% RSLogix 500 project Villa_Park_Riverside_Dump_SLC_500_April_16_2021.RSS, saved by version 11.00.00.00 %
PROJECT "AIRDROME"    % processor: type code 8 %

PROGRAM FILES
  LAD 2   52 rungs

DATA FILES
  O0 OUTPUT  2 elements
  I1 INPUT  3 elements
  S2 STATUS  16 elements
  B3 BINARY  3 elements
  T4 TIMER  15 elements
  C5 COUNTER  1 elements
  R6 CONTROL  1 elements
  N7 INTEGER  1 elements

LADDER 2
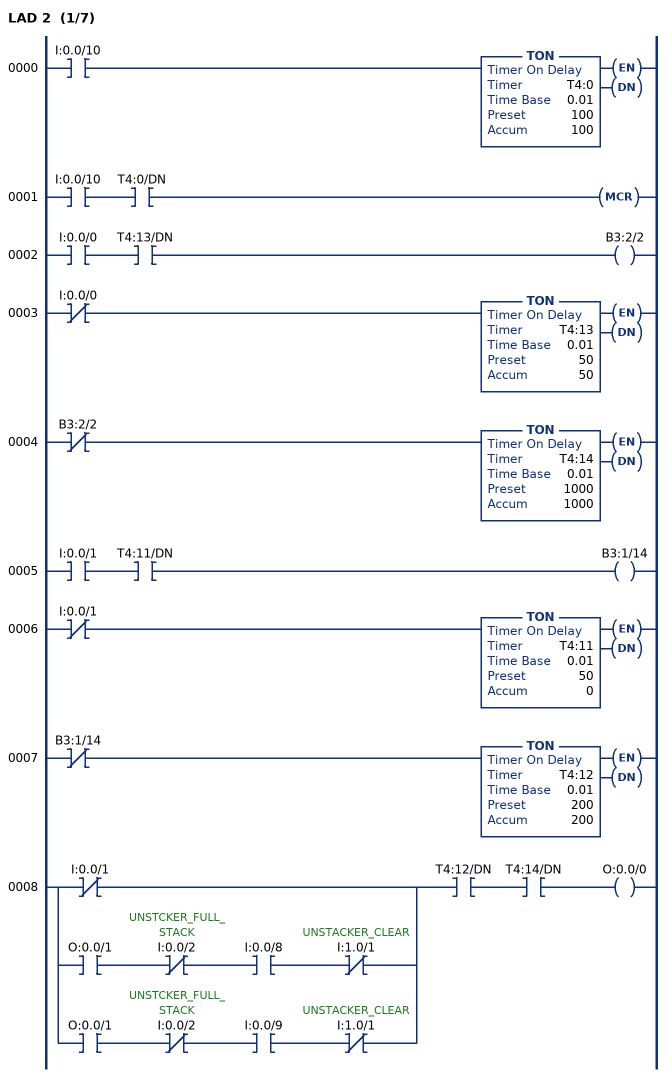
% Rung: 0 %
SOR XIC I:0.0/10 TON T4:0 0.01 100 100 EOR
% Rung: 1 %
SOR XIC I:0.0/10 XIC T4:0/DN MCR EOR
% Rung: 2 %
SOR XIC I:0.0/0 XIC T4:13/DN OTE B3:2/2 EOR
% Rung: 3 %
SOR XIO I:0.0/0 TON T4:13 0.01 50 50 EOR
% Rung: 4 %
SOR XIO B3:2/2 TON T4:14 0.01 1000 1000 EOR
% Rung: 5 %
SOR XIC I:0.0/1 XIC T4:11/DN OTE B3:1/14 EOR
% Rung: 6 %
SOR XIO I:0.0/1 TON T4:11 0.01 50 0 EOR
% Rung: 7 %
SOR XIO B3:1/14 TON T4:12 0.01 200 200 EOR
% Rung: 8 %
SOR BST XIO I:0.0/1 NXB XIC O:0.0/1 XIO I:0.0/2 XIC I:0.0/8 XIO I:1.0/1 NXB XIC O:0.0/1 XIO I:0.0/2 XIC I:0.0/9 XIO I:1.0/1 BND XIC T4:12/DN XIC T4:14/DN OTE O:0.0/0 EOR
%   I:0.0/2  UNSTCKER_FULL_STACK %
%   I:1.0/1  UNSTACKER_CLEAR %

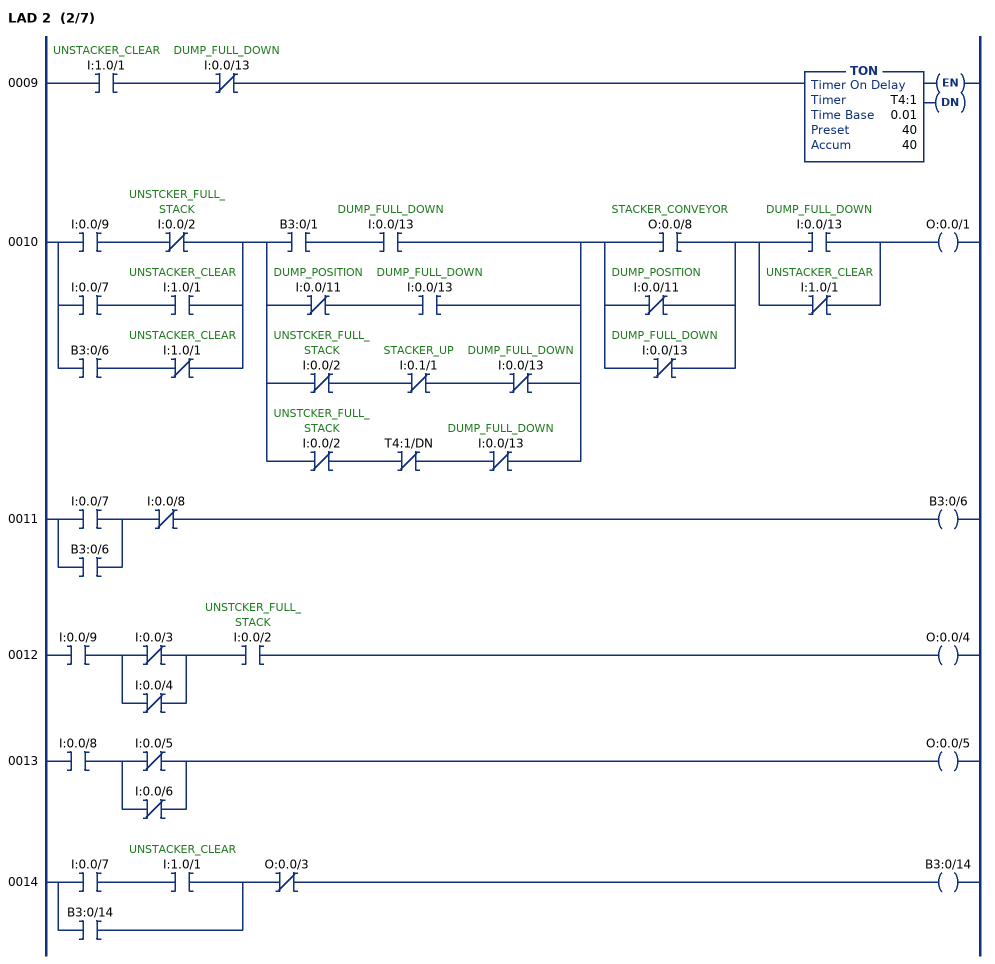
% Rung: 9 %
SOR XIC I:1.0/1 XIO I:0.0/13 TON T4:1 0.01 40 40 EOR
%   I:1.0/1  UNSTACKER_CLEAR %
%   I:0.0/13  DUMP_FULL_DOWN %
% Rung: 10 %
SOR BST XIC I:0.0/9 XIO I:0.0/2 NXB XIC I:0.0/7 XIC I:1.0/1 NXB XIC B3:0/6 XIO I:1.0/1 BND BST XIC B3:0/1 XIC I:0.0/13 NXB XIO I:0.0/11 XIC I:0.0/13 NXB XIO I:0.0/2 XIO I:0.1/1 XIO I:0.0/13 NXB XIO I:0.0/2 XIO T4:1/DN XIO I:0.0/13 BND BST XIC O:0.0/8 NXB XIO I:0.0/11 NXB XIO I:0.0/13 BND BST XIC I:0.0/13 NXB XIO I:1.0/1 BND OTE O:0.0/1 EOR
%   I:0.0/2  UNSTCKER_FULL_STACK %
%   I:1.0/1  UNSTACKER_CLEAR %
%   I:0.0/13  DUMP_FULL_DOWN %
%   I:0.0/11  DUMP_POSITION %
%   I:0.1/1  STACKER_UP %
%   O:0.0/8  STACKER_CONVEYOR %
% Rung: 11 %
SOR BST XIC I:0.0/7 NXB XIC B3:0/6 BND XIO I:0.0/8 OTE B3:0/6 EOR
% Rung: 12 %
SOR XIC I:0.0/9 BST XIO I:0.0/3 NXB XIO I:0.0/4 BND XIC I:0.0/2 OTE O:0.0/4 EOR
%   I:0.0/2  UNSTCKER_FULL_STACK %
% Rung: 13 %
SOR XIC I:0.0/8 BST XIO I:0.0/5 NXB XIO I:0.0/6 BND OTE O:0.0/5 EOR
% Rung: 14 %
SOR BST XIC I:0.0/7 XIC I:1.0/1 NXB XIC B3:0/14 BND XIO O:0.0/3 OTE B3:0/14 EOR
%   I:1.0/1  UNSTACKER_CLEAR %

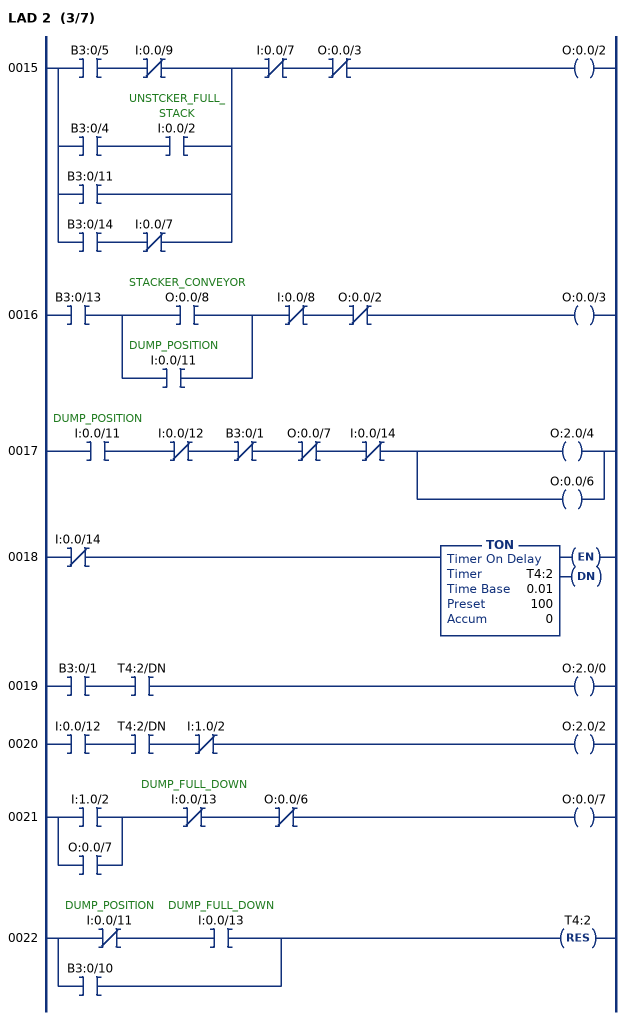
% Rung: 15 %
SOR BST XIC B3:0/5 XIO I:0.0/9 NXB XIC B3:0/4 XIC I:0.0/2 NXB XIC B3:0/11 NXB XIC B3:0/14 XIO I:0.0/7 BND XIO I:0.0/7 XIO O:0.0/3 OTE O:0.0/2 EOR
%   I:0.0/2  UNSTCKER_FULL_STACK %
% Rung: 16 %
SOR XIC B3:0/13 BST XIC O:0.0/8 NXB XIC I:0.0/11 BND XIO I:0.0/8 XIO O:0.0/2 OTE O:0.0/3 EOR
%   O:0.0/8  STACKER_CONVEYOR %
%   I:0.0/11  DUMP_POSITION %
% Rung: 17 %
SOR XIC I:0.0/11 XIO I:0.0/12 XIO B3:0/1 XIO O:0.0/7 XIO I:0.0/14 BST OTE O:2.0/4 NXB OTE O:0.0/6 BND EOR
%   I:0.0/11  DUMP_POSITION %
% Rung: 18 %
SOR XIO I:0.0/14 TON T4:2 0.01 100 0 EOR
% Rung: 19 %
SOR XIC B3:0/1 XIC T4:2/DN OTE O:2.0/0 EOR
% Rung: 20 %
SOR XIC I:0.0/12 XIC T4:2/DN XIO I:1.0/2 OTE O:2.0/2 EOR
% Rung: 21 %
SOR BST XIC I:1.0/2 NXB XIC O:0.0/7 BND XIO I:0.0/13 XIO O:0.0/6 OTE O:0.0/7 EOR
%   I:0.0/13  DUMP_FULL_DOWN %
% Rung: 22 %
SOR BST XIO I:0.0/11 XIC I:0.0/13 NXB XIC B3:0/10 BND RES T4:2 EOR
%   I:0.0/11  DUMP_POSITION %
%   I:0.0/13  DUMP_FULL_DOWN %

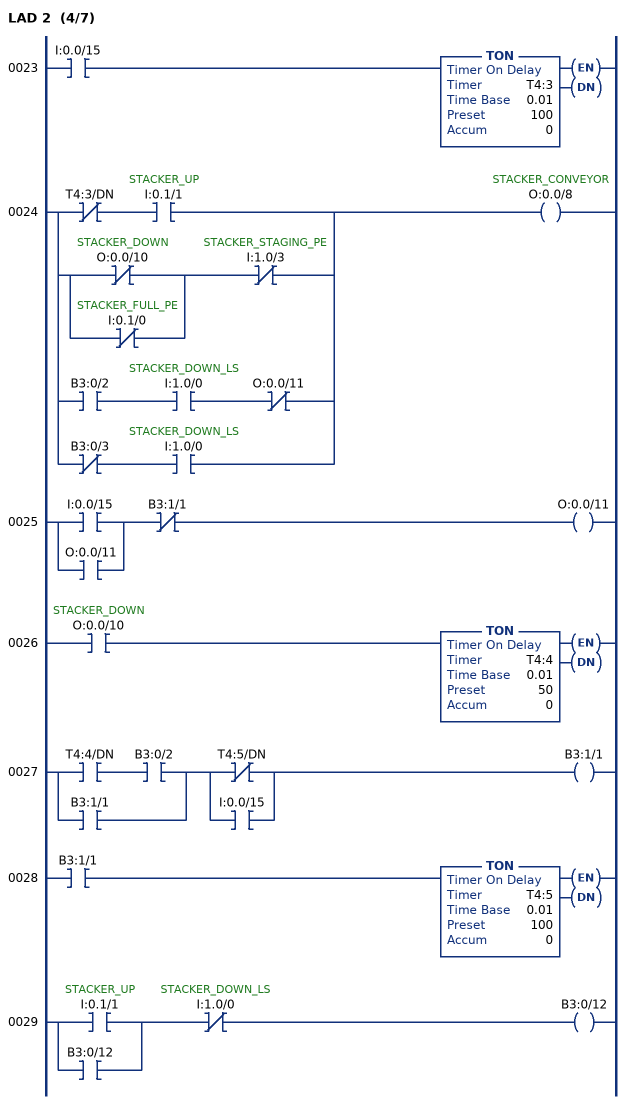
% Rung: 23 %
SOR XIC I:0.0/15 TON T4:3 0.01 100 0 EOR
% Rung: 24 %
SOR BST BST XIO T4:3/DN XIC I:0.1/1 NXB BST XIO O:0.0/10 NXB XIO I:0.1/0 BND XIO I:1.0/3 BND NXB XIC B3:0/2 XIC I:1.0/0 XIO O:0.0/11 NXB XIO B3:0/3 XIC I:1.0/0 BND OTE O:0.0/8 EOR
%   I:0.1/1  STACKER_UP %
%   O:0.0/10  STACKER_DOWN %
%   I:0.1/0  STACKER_FULL_PE %
%   I:1.0/3  STACKER_STAGING_PE %
%   I:1.0/0  STACKER_DOWN_LS %
%   O:0.0/8  STACKER_CONVEYOR %
% Rung: 25 %
SOR BST XIC I:0.0/15 NXB XIC O:0.0/11 BND XIO B3:1/1 OTE O:0.0/11 EOR
% Rung: 26 %
SOR XIC O:0.0/10 TON T4:4 0.01 50 0 EOR
%   O:0.0/10  STACKER_DOWN %
% Rung: 27 %
SOR BST XIC T4:4/DN XIC B3:0/2 NXB XIC B3:1/1 BND BST XIO T4:5/DN NXB XIC I:0.0/15 BND OTE B3:1/1 EOR
% Rung: 28 %
SOR XIC B3:1/1 TON T4:5 0.01 100 0 EOR
% Rung: 29 %
SOR BST XIC I:0.1/1 NXB XIC B3:0/12 BND XIO I:1.0/0 OTE B3:0/12 EOR
%   I:0.1/1  STACKER_UP %
%   I:1.0/0  STACKER_DOWN_LS %

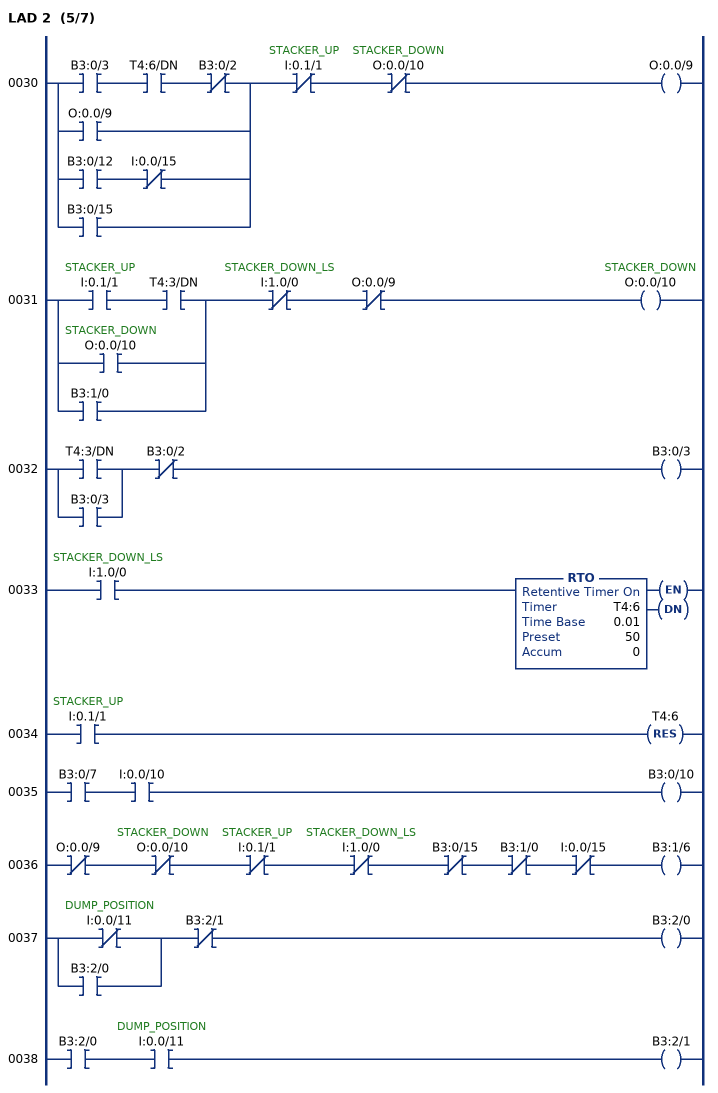
% Rung: 30 %
SOR BST XIC B3:0/3 XIC T4:6/DN XIO B3:0/2 NXB XIC O:0.0/9 NXB XIC B3:0/12 XIO I:0.0/15 NXB XIC B3:0/15 BND XIO I:0.1/1 XIO O:0.0/10 OTE O:0.0/9 EOR
%   I:0.1/1  STACKER_UP %
%   O:0.0/10  STACKER_DOWN %
% Rung: 31 %
SOR BST XIC I:0.1/1 XIC T4:3/DN NXB XIC O:0.0/10 NXB XIC B3:1/0 BND XIO I:1.0/0 XIO O:0.0/9 OTE O:0.0/10 EOR
%   I:0.1/1  STACKER_UP %
%   O:0.0/10  STACKER_DOWN %
%   I:1.0/0  STACKER_DOWN_LS %
% Rung: 32 %
SOR BST XIC T4:3/DN NXB XIC B3:0/3 BND XIO B3:0/2 OTE B3:0/3 EOR
% Rung: 33 %
SOR XIC I:1.0/0 RTO T4:6 0.01 50 0 EOR
%   I:1.0/0  STACKER_DOWN_LS %
% Rung: 34 %
SOR XIC I:0.1/1 RES T4:6 EOR
%   I:0.1/1  STACKER_UP %
% Rung: 35 %
SOR XIC B3:0/7 XIC I:0.0/10 OTE B3:0/10 EOR
% Rung: 36 %
SOR XIO O:0.0/9 XIO O:0.0/10 XIO I:0.1/1 XIO I:1.0/0 XIO B3:0/15 XIO B3:1/0 XIO I:0.0/15 OTE B3:1/6 EOR
%   O:0.0/10  STACKER_DOWN %
%   I:0.1/1  STACKER_UP %
%   I:1.0/0  STACKER_DOWN_LS %
% Rung: 37 %
SOR BST XIO I:0.0/11 NXB XIC B3:2/0 BND XIO B3:2/1 OTE B3:2/0 EOR
%   I:0.0/11  DUMP_POSITION %
% Rung: 38 %
SOR XIC B3:2/0 XIC I:0.0/11 OTE B3:2/1 EOR
%   I:0.0/11  DUMP_POSITION %

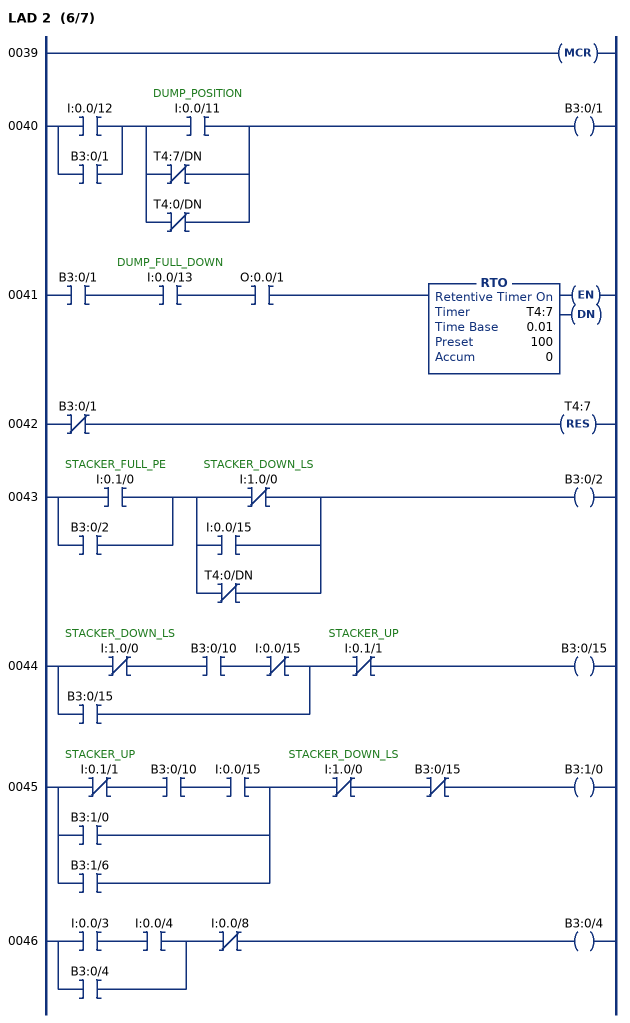
% Rung: 39 %
SOR MCR EOR
% Rung: 40 %
SOR BST XIC I:0.0/12 NXB XIC B3:0/1 BND BST XIC I:0.0/11 NXB XIO T4:7/DN NXB XIO T4:0/DN BND OTE B3:0/1 EOR
%   I:0.0/11  DUMP_POSITION %
% Rung: 41 %
SOR XIC B3:0/1 XIC I:0.0/13 XIC O:0.0/1 RTO T4:7 0.01 100 0 EOR
%   I:0.0/13  DUMP_FULL_DOWN %
% Rung: 42 %
SOR XIO B3:0/1 RES T4:7 EOR
% Rung: 43 %
SOR BST XIC I:0.1/0 NXB XIC B3:0/2 BND BST XIO I:1.0/0 NXB XIC I:0.0/15 NXB XIO T4:0/DN BND OTE B3:0/2 EOR
%   I:0.1/0  STACKER_FULL_PE %
%   I:1.0/0  STACKER_DOWN_LS %
% Rung: 44 %
SOR BST XIO I:1.0/0 XIC B3:0/10 XIO I:0.0/15 NXB XIC B3:0/15 BND XIO I:0.1/1 OTE B3:0/15 EOR
%   I:1.0/0  STACKER_DOWN_LS %
%   I:0.1/1  STACKER_UP %
% Rung: 45 %
SOR BST XIO I:0.1/1 XIC B3:0/10 XIC I:0.0/15 NXB XIC B3:1/0 NXB XIC B3:1/6 BND XIO I:1.0/0 XIO B3:0/15 OTE B3:1/0 EOR
%   I:0.1/1  STACKER_UP %
%   I:1.0/0  STACKER_DOWN_LS %
% Rung: 46 %
SOR BST XIC I:0.0/3 XIC I:0.0/4 NXB XIC B3:0/4 BND XIO I:0.0/8 OTE B3:0/4 EOR

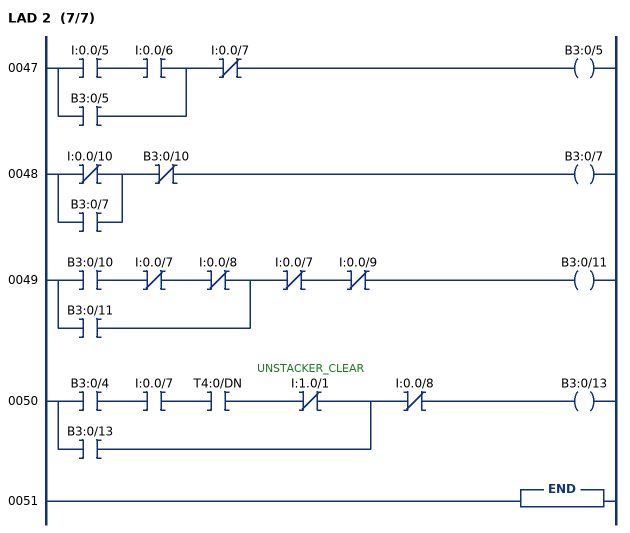
% Rung: 47 %
SOR BST XIC I:0.0/5 XIC I:0.0/6 NXB XIC B3:0/5 BND XIO I:0.0/7 OTE B3:0/5 EOR
% Rung: 48 %
SOR BST XIO I:0.0/10 NXB XIC B3:0/7 BND XIO B3:0/10 OTE B3:0/7 EOR
% Rung: 49 %
SOR BST XIC B3:0/10 XIO I:0.0/7 XIO I:0.0/8 NXB XIC B3:0/11 BND XIO I:0.0/7 XIO I:0.0/9 OTE B3:0/11 EOR
% Rung: 50 %
SOR BST XIC B3:0/4 XIC I:0.0/7 XIC T4:0/DN XIO I:1.0/1 NXB XIC B3:0/13 BND XIO I:0.0/8 OTE B3:0/13 EOR
%   I:1.0/1  UNSTACKER_CLEAR %
% Rung: 51 %
SOR END EOR

DATA TABLE (non-zero values as saved)
DATA B3
% B3:0 % 0X1028 0X0000 0X0000
DATA T4
% .PRE .ACC %
% T4:0 % 100 100
% T4:1 % 40 40
% T4:2 % 100 0
% T4:3 % 100 0
% T4:4 % 50 0
% T4:5 % 100 0
% T4:6 % 50 0
% T4:7 % 100 0
% T4:8 % 100 0
% T4:10 % 2500 0
% T4:11 % 50 0
% T4:12 % 200 200
% T4:13 % 50 50
% T4:14 % 1000 1000
